// TIA Portal V19 program export: 1 tag tables, 0 data types, 1 data blocks, 1 code blocks (in call order from the OBs), 2 instance data blocks

VAR_GLOBAL   // PLC tag table "Default tag table"
   System_Byte AT %MB1 : Byte;
   FirstScan AT %M1.0 : Bool;
   DiagStatusUpdate AT %M1.1 : Bool;
   AlwaysTRUE AT %M1.2 : Bool;
   AlwaysFALSE AT %M1.3 : Bool;
   Clock_Byte AT %MB0 : Byte;
   Clock_10Hz AT %M0.0 : Bool;
   Clock_5Hz AT %M0.1 : Bool;
   "Clock_2.5Hz" AT %M0.2 : Bool;
   Clock_2Hz AT %M0.3 : Bool;
   "Clock_1.25Hz" AT %M0.4 : Bool;
   Clock_1Hz AT %M0.5 : Bool;
   "Clock_0.625Hz" AT %M0.6 : Bool;
   "Clock_0.5Hz" AT %M0.7 : Bool;
   Encoder_HSC_Count AT %ID1000 : DInt;
   Ch_A AT %I0.0 : Bool;
   Ch_B AT %I0.1 : Bool;
   Reset_Btn AT %I0.2 : Bool;
   Max_Len_Pos_Edg_Mem AT %M2.0 : Bool;
END_VAR

DATA_BLOCK "Measurement_Data"   // DB2
{ S7_Optimized_Access := 'FALSE' }
   VAR RETAIN
      Length : Real;
      Last_Measurement : Real;
      Encoder_Cnt : DInt;
      Pulses_Per_Meter : DInt := 2048;
      Reset : Bool;
      Data_Logger_Bit : Bool;
   END_VAR
BEGIN
END_DATA_BLOCK

ORGANIZATION_BLOCK "Main"   // OB1, LAD, ProgramCycle
TITLE = "Main Program Sweep (Cycle)"
{ S7_Optimized_Access := 'TRUE' }
// stored: SetENOAutomatically false
   VAR_INPUT
      Initial_Call : Bool;   // Initial call of this OB
      Remanence : Bool;   // =True, if remanent data are available
   END_VAR
   VAR_TEMP   // added for the SCL form of the ladder/FBD networks
      _w1 : Bool;
   END_VAR
BEGIN

REGION Network 1
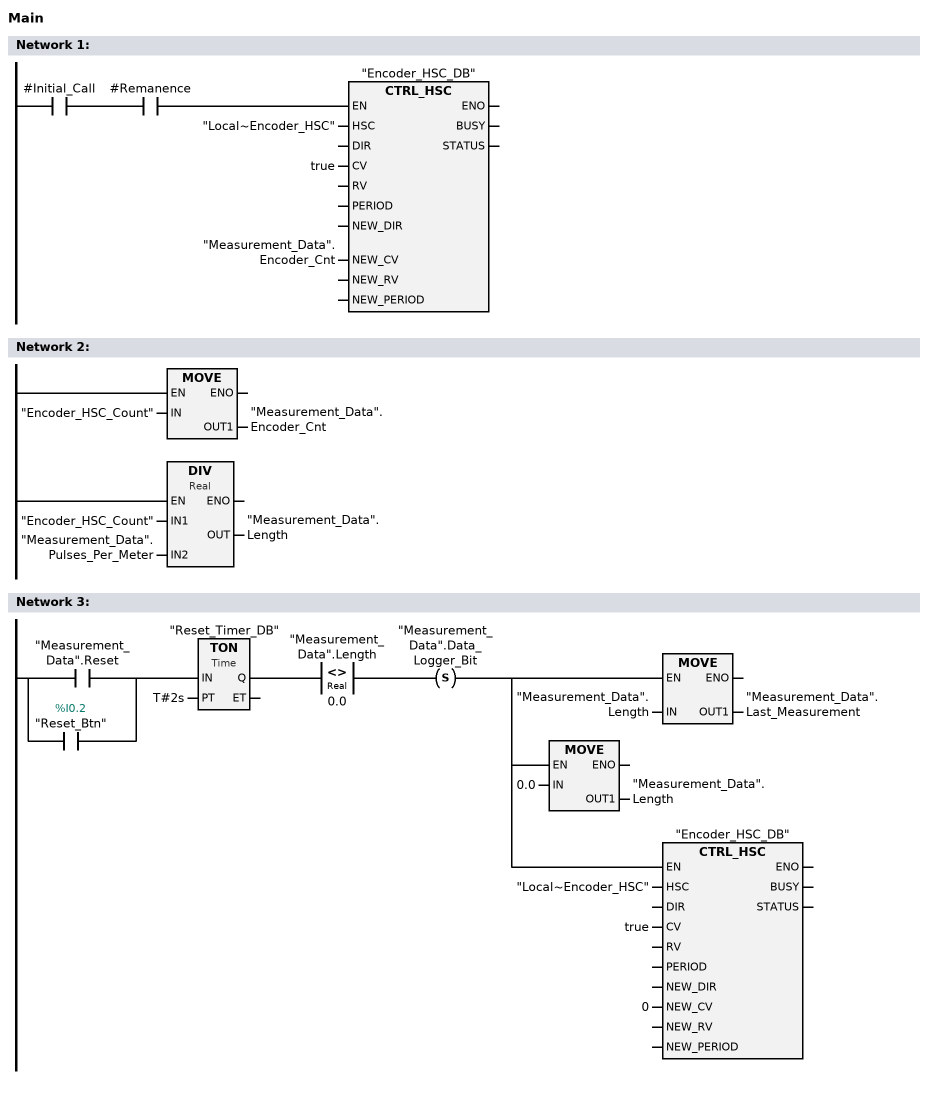
   RUNG wire#powerrail
      Contact( #Initial_Call )
      Contact( #Remanence )
      "Encoder_HSC_DB".CTRL_HSC(HSC := "Local~Encoder_HSC", DIR :=, CV := true, RV :=, PERIOD :=, NEW_DIR :=, NEW_CV := "Measurement_Data".Encoder_Cnt, NEW_RV :=, NEW_PERIOD :=, BUSY =>, STATUS =>)
   END_RUNG
   // the same network as SCL:
   IF #Initial_Call AND #Remanence THEN
       "Encoder_HSC_DB"(HSC := "Local~Encoder_HSC", CV := true, NEW_CV := "Measurement_Data".Encoder_Cnt);   // CTRL_HSC
   END_IF;
END_REGION

REGION Network 2
   RUNG wire#powerrail
      Move(in := "Encoder_HSC_Count", out1 => "Measurement_Data".Encoder_Cnt)
   END_RUNG
   RUNG wire#powerrail
      { S7_Templates := "SrcType := Real" } Div(in1 := "Encoder_HSC_Count", in2 := "Measurement_Data".Pulses_Per_Meter, out => "Measurement_Data".Length)
   END_RUNG
   // the same network as SCL:
   "Measurement_Data".Encoder_Cnt := "Encoder_HSC_Count";
   "Measurement_Data".Length := "Encoder_HSC_Count" / "Measurement_Data".Pulses_Per_Meter;
END_REGION

REGION Network 3
   RUNG wire#powerrail
      Contact( "Measurement_Data".Reset )
      wire#w1
      { S7_Templates := "time_type := Time" } "Reset_Timer_DB".TON(pt := T#2s, et =>)
      { S7_Templates := "SrcType := Real" } NE_Contact(in1 := "Measurement_Data".Length, in2 := 0.0)
      S_Coil( "Measurement_Data".Data_Logger_Bit )
      wire#w2
      Move(in := "Measurement_Data".Length, out1 => "Measurement_Data".Last_Measurement)
   END_RUNG
   RUNG wire#powerrail
      Contact( "Reset_Btn" )
   END_RUNG wire#w1
   RUNG wire#w2
      Move(in := 0.0, out1 => "Measurement_Data".Length)
   END_RUNG
   RUNG wire#w2
      "Encoder_HSC_DB".CTRL_HSC(HSC := "Local~Encoder_HSC", DIR :=, CV := true, RV :=, PERIOD :=, NEW_DIR :=, NEW_CV := 0, NEW_RV :=, NEW_PERIOD :=, BUSY =>, STATUS =>)
   END_RUNG
   // the same network as SCL:
   "Reset_Timer_DB".TON(IN := "Measurement_Data".Reset OR "Reset_Btn", PT := T#2s);
   IF "Reset_Timer_DB".Q AND ("Measurement_Data".Length <> 0.0) THEN
       "Measurement_Data".Data_Logger_Bit := TRUE;
       "Measurement_Data".Last_Measurement := "Measurement_Data".Length;
   END_IF;
   #_w1 := "Reset_Timer_DB".Q AND ("Measurement_Data".Length <> 0.0);
   IF #_w1 THEN
       "Measurement_Data".Length := 0.0;
       "Encoder_HSC_DB"(HSC := "Local~Encoder_HSC", CV := true, NEW_CV := 0);   // CTRL_HSC
   END_IF;
END_REGION
END_ORGANIZATION_BLOCK

DATA_BLOCK "Encoder_HSC_DB"   // DB1
// stored: InstanceOfName CTRL_HSC, OfSystemLibElement CTRL_HSC, OfSystemLibVersion 1.0
"CTRL_HSC"
   // VAR_INPUT
   //    HSC : HW_HSC;
   //    DIR : Bool;
   //    CV : Bool;
   //    RV : Bool;
   //    PERIOD : Bool;
   //    NEW_DIR : Int;
   //    NEW_CV : DInt;
   //    NEW_RV : DInt;
   //    NEW_PERIOD : Int;
   // END_VAR
   // VAR_OUTPUT
   //    BUSY : Bool;
   //    STATUS : Word;
   // END_VAR
BEGIN
END_DATA_BLOCK

DATA_BLOCK "Reset_Timer_DB"   // DB3
{ S7_Optimized_Access := 'TRUE' }
// stored: InstanceOfName IEC_TIMER, OfSystemLibElement IEC_TIMER, OfSystemLibVersion 1.0
"IEC_TIMER"
   // VAR
   //    PT : Time;
   //    ET { ExternalWritable := 'False'} : Time;
   //    IN : Bool;
   //    Q { ExternalWritable := 'False'} : Bool;
   // END_VAR
BEGIN
END_DATA_BLOCK
